FUNCTION_BLOCK FB_ProBoxElementVC_Base EXTENDS FB_ElementMpdBase
VAR_INPUT
END_VAR
VAR_OUTPUT
END_VAR
VAR
END_VAR

METHOD PROTECTED _M_CheckErrors : BOOL
VAR_IN_OUT
	MpdExternalErrors					: ST_MPD_ExternalErrors;
	SgGroupRef							: FB_ProBOXSG;	//Reference to Switching group
END_VAR
VAR
	i:INT;
	UserMsg	: STRING(System.ERROR_PARAM_STRINGLENGTH) := 'Check door at level: ';
END_VAR

F_ResetError(FALSE, ElementData.ErrorData.ErrorDataSet[3]);


// ----------------------------------------------------
// Normally open errors
// ----------------------------------------------------

//Set error if Error hi temp lift resistor
IF MpdExternalErrors.HighTempResLift THEN
	
		F_SetError(	
			ErrorType	:= E_ErrorType.ERROR,
			ErrorParam	:= 'Hi temp lift resistor',
			ErrorMsg	:= E_ErrorConv.DRIVE_ERROR,
			ErrorData	:= ElementData.ErrorData.ErrorDataSet[3]);	
END_IF

//Set error if Error hi temp drive resistor
IF MpdExternalErrors.HighTempResDrive THEN
	
		F_SetError(	
			ErrorType	:= E_ErrorType.ERROR,
			ErrorParam	:= 'Hi temp drive resistor',
			ErrorMsg	:= E_ErrorConv.DRIVE_ERROR,
			ErrorData	:= ElementData.ErrorData.ErrorDataSet[3]);	
END_IF

//Set error if FrequencyInverterError
IF MpdExternalErrors.FrequencyInverterError THEN
	
		F_SetError(	
			ErrorType	:= E_ErrorType.ERROR,
			ErrorParam	:= 'VC Freqency inverter',
			ErrorMsg	:= E_ErrorConv.DRIVE_ERROR,
			ErrorData	:= ElementData.ErrorData.ErrorDataSet[3]);
END_IF

// ----------------------------------------------------
// Normally closed errors
// ----------------------------------------------------

//Set error if Error from the belts (Slackwire)
IF NOT MpdExternalErrors.BeltMonitoring THEN
	
		F_SetError(	
			ErrorType	:= E_ErrorType.ERROR,
			ErrorParam	:= 'Belt Monitoring Error',
			ErrorMsg	:= E_ErrorConv.LIMIT_SWITCH_ACTIVE,
			ErrorData	:= ElementData.ErrorData.ErrorDataSet[3]);	
END_IF

//Set error if FallBrake occurres
IF NOT MpdExternalErrors.FallBrake  THEN	
	F_SetError(	
			ErrorType	:= E_ErrorType.ERROR,
			ErrorParam	:= 'FallBrake Has Occurred',
			ErrorMsg	:= E_ErrorConv.LIMIT_SWITCH_ACTIVE,
			ErrorData	:= ElementData.ErrorData.ErrorDataSet[3]);	
END_IF

IF NOT MpdExternalErrors.FallBrakeSpeedRegulator THEN	
	F_SetError(	
			ErrorType	:= E_ErrorType.ERROR,
			ErrorParam	:= 'FallBrake Speedregulator',
			ErrorMsg	:= E_ErrorConv.LIMIT_SWITCH_ACTIVE,
			ErrorData	:= ElementData.ErrorData.ErrorDataSet[3]);	
END_IF

IF NOT MpdExternalErrors.SlackWire THEN	
	F_SetError(	
			ErrorType	:= E_ErrorType.ERROR,
			ErrorParam	:= 'Slack wire limit switch',
			ErrorMsg	:= E_ErrorConv.LIMIT_SWITCH_ACTIVE,
			ErrorData	:= ElementData.ErrorData.ErrorDataSet[3]);	
END_IF


//Check doors
FOR i:=1 TO 32 DO
	
	IF( NOT MpdExternalErrors.DoorClosedLevel[i]) THEN
		UserMsg := CONCAT(UserMsg,TO_STRING(i));
		F_SetError(	
				ErrorType	:= E_ErrorType.ERROR,
				ErrorParam	:= UserMsg,
				ErrorMsg	:= E_ErrorConv.DOOR_ERROR,
				ErrorData	:= ElementData.ErrorData.ErrorDataSet[3]);	
	END_IF
END_FOR


SUPER^._M_CheckMpdErrors(MpdExternalErrors.EndLimit,MpdExternalErrors.HighTempResDrive, SgGroupRef, ElementData.ErrorData.ErrorDataSet[3]);
END_METHOD

//TS panel and Access panel on for same maintenance level works in conjunction with eachother. An TS panel start button can cancel AP panel Entry Request 
METHOD PUBLIC M_PowerStoreEntry : BOOL
VAR_INPUT
	AccessPanel_Index		: INT; 	// Access panel (Level entrance panel) index
	TS_Panel_Index			: INT; 	// Transfer Station panel index	
	AbortEntryReq			: BOOL;	// TRUE = Abort a entry request (typically a start button from TS panel will abort a entry request from AP panel)
	TS_Panel_EntryReq		: BOOL; // TRUE = Make a entry request from an TS panel
END_VAR

//Abort Access panel entry request if gate is closed.
fbEntryRequestCtrl.M_AbortEntryRequest(AccessPanel_Index, AbortEntryReq);

// register the entry request from an TS panel.
fbEntryRequestCtrl.M_RegisterEntryRequest(TS_Panel_EntryReq,TS_Panel_Index);
END_METHOD

//Option to apply external condition for desition if the entry is safe for the operator.
METHOD PUBLIC M_RequestEntryExtDev : BOOL
VAR_INPUT
	WaitForExternalDevice	: BOOL;		// wait in Entry pending state for an external device
	CabinetIndex			: INT;		// the index of the cabinet
END_VAR

fbEntryRequestCtrl.M_WaitForExternalDevice(WaitForExternalDevice,CabinetIndex);
END_METHOD

METHOD PUBLIC M_SetHeightCorrection : BOOL
VAR_INPUT
	PickupCondition	: BOOL;		//Condition to start Pickup height compensation
	DepositCondition : BOOL;	//Condition to start deposit height compensation
	PickupAdjustment : INT;		//Height to compensate when pickup or deposit. positive or negative value [mm]
	DepositAdjustment : INT;	//Height to compensate when pickup or deposit. positive or negative value [mm]	
END_VAR

fbMpdControl.P_AutoAdjustVcHeight.PickupCondition	:= PickupCondition;
fbMpdControl.P_AutoAdjustVcHeight.DepositCondition	:= DepositCondition;
fbMpdControl.P_AutoAdjustVcHeight.PickupAdjustment	:= PickupAdjustment;
fbMpdControl.P_AutoAdjustVcHeight.DepositAdjustment 	:= DepositAdjustment;
END_METHOD

END_FUNCTION_BLOCK

(* stored: Version 1.1.0.1, ProductVersion 3.1.4024.9
   POU FB_ProBoxElementVC_Base: Id {97508358-d381-4a45-b82f-e0e4c8802e3c}, SpecialFunc None
   Method _M_CheckErrors: Id {d9e22ad7-1aa5-413e-b121-68627c1f3574}
   Method M_PowerStoreEntry: Id {2479ecf2-f632-49df-b3fb-f10e1e7c84ef}
   Method M_RequestEntryExtDev: Id {e435af44-b13b-4e95-b7a5-48b0cc229984}
   Method M_SetHeightCorrection: Id {66cc9226-a8c0-41c9-8ba2-9611861292e5} *)
